// TIA Portal V17 export
// export: Created 2025-03-07T09:17:46.2678876Z, ExportSetting WithDefaults, DisplayName Totally Integrated Automation Portal, DisplayVersion V17 Update 8, DisplayName TIA Portal Openness, DisplayVersion V17 Update 8, DisplayName TIA Portal Version Control Interface, DisplayVersion V17, DisplayName SINAMICS Startdrive Advanced, DisplayVersion V17 SP2, DisplayName SINAMICS Startdrive G110M, G120, G120C, G120D, G120P, G115D, DisplayVersion V17 SP2, DisplayName SINAMICS Startdrive G130, G150, S120, S150, SINAMICS MV, S210, DisplayVersion V17 SP2, DisplayName STEP 7 Professional, DisplayVersion V17 Update 8, DisplayName SINUMERIK ONE STEP 7 Toolbox, DisplayVersion V17 Update 12, DisplayName SINUMERIK 840D sl STEP 7 Toolbox, DisplayVersion V17 Update 12, DisplayName STEP 7 Safety, DisplayVersion V17 Update 6, DisplayName WinCC Advanced, DisplayVersion V17 Update 8
FUNCTION "FC2107_MACHINE_LIGHT" : Void   // FC2107, LAD
{ S7_Optimized_Access := 'FALSE' }
AUTHOR : ETXETAR
VERSION : 1.0
// stored: AutoNumber false, IsIECCheckEnabled false, SetENOAutomatically false, UDAEnableTagReadback false
   VAR_TEMP   // added for the SCL form of the ladder/FBD networks
      _w1 : Bool;
      _w2 : Bool;
      _w3 : Bool;
      _w4 : Bool;
   END_VAR
BEGIN

REGION Network 1: INPUTS
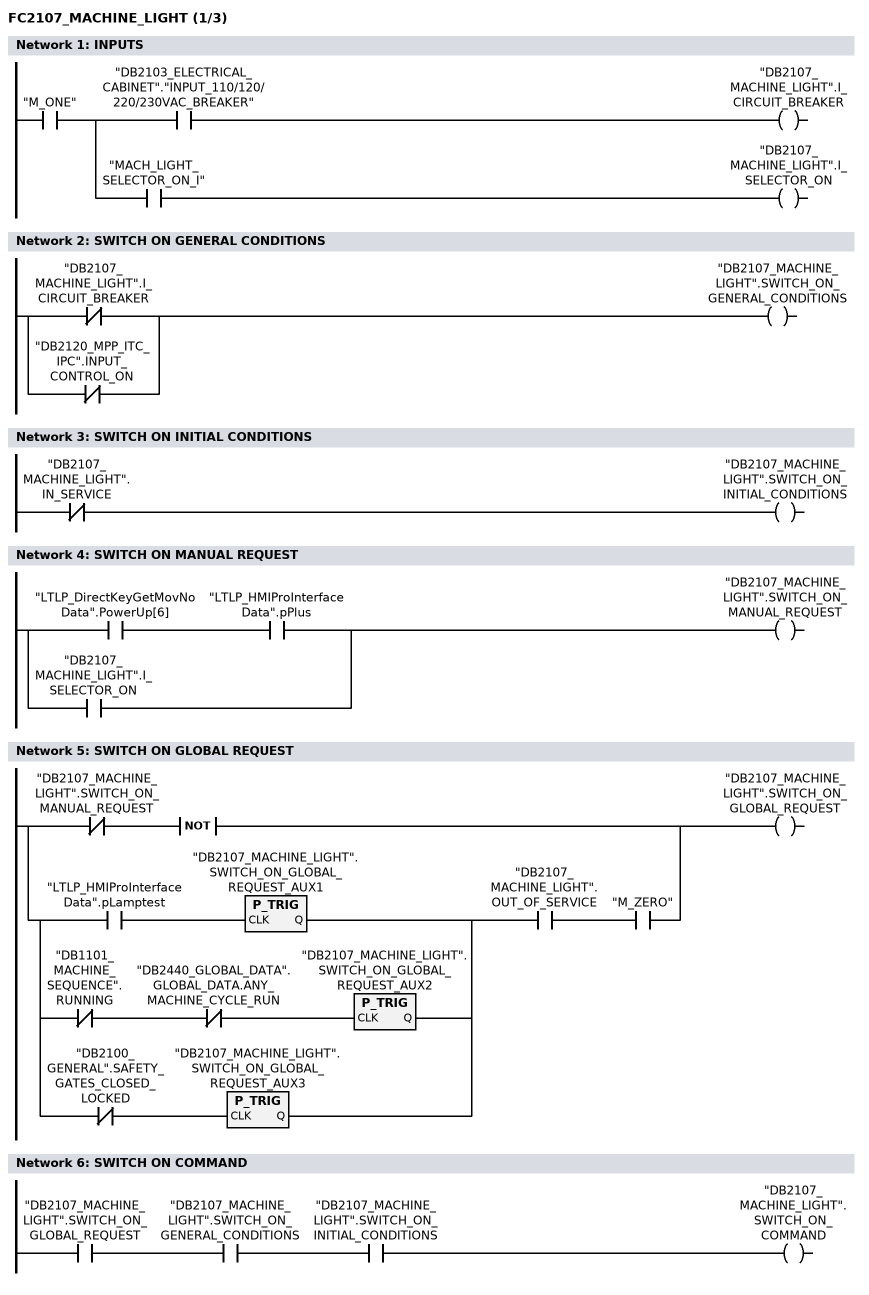
   RUNG wire#powerrail
      Contact( "M_ONE" )
      wire#w1
      Contact( "DB2103_ELECTRICAL_CABINET"."INPUT_110/120/220/230VAC_BREAKER" )
      Coil( "DB2107_MACHINE_LIGHT".I_CIRCUIT_BREAKER )
   END_RUNG
   RUNG wire#w1
      Contact( "MACH_LIGHT_SELECTOR_ON_I" )
      Coil( "DB2107_MACHINE_LIGHT".I_SELECTOR_ON )
   END_RUNG
   // the same network as SCL:
   "DB2107_MACHINE_LIGHT".I_CIRCUIT_BREAKER := "M_ONE" AND "DB2103_ELECTRICAL_CABINET"."INPUT_110/120/220/230VAC_BREAKER";
   "DB2107_MACHINE_LIGHT".I_SELECTOR_ON := "M_ONE" AND "MACH_LIGHT_SELECTOR_ON_I";
END_REGION

REGION Network 2: SWITCH ON GENERAL CONDITIONS
   RUNG wire#powerrail
      I_Contact( "DB2107_MACHINE_LIGHT".I_CIRCUIT_BREAKER )
      wire#w1
      Coil( "DB2107_MACHINE_LIGHT".SWITCH_ON_GENERAL_CONDITIONS )
   END_RUNG
   RUNG wire#powerrail
      I_Contact( "DB2120_MPP_ITC_IPC".INPUT_CONTROL_ON )
   END_RUNG wire#w1
   // the same network as SCL:
   "DB2107_MACHINE_LIGHT".SWITCH_ON_GENERAL_CONDITIONS := NOT "DB2107_MACHINE_LIGHT".I_CIRCUIT_BREAKER OR NOT "DB2120_MPP_ITC_IPC".INPUT_CONTROL_ON;
END_REGION

REGION Network 3: SWITCH ON INITIAL CONDITIONS
   RUNG wire#powerrail
      I_Contact( "DB2107_MACHINE_LIGHT".IN_SERVICE )
      Coil( "DB2107_MACHINE_LIGHT".SWITCH_ON_INITIAL_CONDITIONS )
   END_RUNG
   // the same network as SCL:
   "DB2107_MACHINE_LIGHT".SWITCH_ON_INITIAL_CONDITIONS := NOT "DB2107_MACHINE_LIGHT".IN_SERVICE;
END_REGION

REGION Network 4: SWITCH ON MANUAL REQUEST
   RUNG wire#powerrail
      Contact( "LTLP_DirectKeyGetMovNoData".PowerUp[6] )
      Contact( "LTLP_HMIProInterfaceData".pPlus )
      wire#w1
      Coil( "DB2107_MACHINE_LIGHT".SWITCH_ON_MANUAL_REQUEST )
   END_RUNG
   RUNG wire#powerrail
      Contact( "DB2107_MACHINE_LIGHT".I_SELECTOR_ON )
   END_RUNG wire#w1
   // the same network as SCL:
   "DB2107_MACHINE_LIGHT".SWITCH_ON_MANUAL_REQUEST := ("LTLP_DirectKeyGetMovNoData".PowerUp[6] AND "LTLP_HMIProInterfaceData".pPlus) OR "DB2107_MACHINE_LIGHT".I_SELECTOR_ON;
END_REGION

REGION Network 5: SWITCH ON GLOBAL REQUEST
   RUNG wire#powerrail
      I_Contact( "DB2107_MACHINE_LIGHT".SWITCH_ON_MANUAL_REQUEST )
      Not()
      wire#w1
      Coil( "DB2107_MACHINE_LIGHT".SWITCH_ON_GLOBAL_REQUEST )
   END_RUNG
   RUNG wire#powerrail
      Contact( "LTLP_HMIProInterfaceData".pLamptest )
      P_Trig( "DB2107_MACHINE_LIGHT".SWITCH_ON_GLOBAL_REQUEST_AUX1 )
      wire#w2
      Contact( "DB2107_MACHINE_LIGHT".OUT_OF_SERVICE )
      Contact( "M_ZERO" )
   END_RUNG wire#w1
   RUNG wire#powerrail
      I_Contact( "DB1101_MACHINE_SEQUENCE".RUNNING )
      I_Contact( "DB2440_GLOBAL_DATA".GLOBAL_DATA.ANY_MACHINE_CYCLE_RUN )
      P_Trig( "DB2107_MACHINE_LIGHT".SWITCH_ON_GLOBAL_REQUEST_AUX2 )
   END_RUNG wire#w2
   RUNG wire#powerrail
      I_Contact( "DB2100_GENERAL".SAFETY_GATES_CLOSED_LOCKED )
      P_Trig( "DB2107_MACHINE_LIGHT".SWITCH_ON_GLOBAL_REQUEST_AUX3 )
   END_RUNG wire#w2
   // the same network as SCL:
   #_w1 := "LTLP_HMIProInterfaceData".pLamptest AND NOT "DB2107_MACHINE_LIGHT".SWITCH_ON_GLOBAL_REQUEST_AUX1;   // rising edge
   "DB2107_MACHINE_LIGHT".SWITCH_ON_GLOBAL_REQUEST_AUX1 := "LTLP_HMIProInterfaceData".pLamptest;
   #_w2 := NOT "DB1101_MACHINE_SEQUENCE".RUNNING AND NOT "DB2440_GLOBAL_DATA".GLOBAL_DATA.ANY_MACHINE_CYCLE_RUN;
   #_w3 := #_w2 AND NOT "DB2107_MACHINE_LIGHT".SWITCH_ON_GLOBAL_REQUEST_AUX2;   // rising edge
   "DB2107_MACHINE_LIGHT".SWITCH_ON_GLOBAL_REQUEST_AUX2 := #_w2;
   #_w4 := NOT "DB2100_GENERAL".SAFETY_GATES_CLOSED_LOCKED AND NOT "DB2107_MACHINE_LIGHT".SWITCH_ON_GLOBAL_REQUEST_AUX3;   // rising edge
   "DB2107_MACHINE_LIGHT".SWITCH_ON_GLOBAL_REQUEST_AUX3 := NOT "DB2100_GENERAL".SAFETY_GATES_CLOSED_LOCKED;
   "DB2107_MACHINE_LIGHT".SWITCH_ON_GLOBAL_REQUEST := NOT (NOT "DB2107_MACHINE_LIGHT".SWITCH_ON_MANUAL_REQUEST) OR ((#_w1 OR #_w3 OR #_w4) AND "DB2107_MACHINE_LIGHT".OUT_OF_SERVICE AND "M_ZERO");
END_REGION

REGION Network 6: SWITCH ON COMMAND
   RUNG wire#powerrail
      Contact( "DB2107_MACHINE_LIGHT".SWITCH_ON_GLOBAL_REQUEST )
      Contact( "DB2107_MACHINE_LIGHT".SWITCH_ON_GENERAL_CONDITIONS )
      Contact( "DB2107_MACHINE_LIGHT".SWITCH_ON_INITIAL_CONDITIONS )
      Coil( "DB2107_MACHINE_LIGHT".SWITCH_ON_COMMAND )
   END_RUNG
   // the same network as SCL:
   "DB2107_MACHINE_LIGHT".SWITCH_ON_COMMAND := "DB2107_MACHINE_LIGHT".SWITCH_ON_GLOBAL_REQUEST AND "DB2107_MACHINE_LIGHT".SWITCH_ON_GENERAL_CONDITIONS AND "DB2107_MACHINE_LIGHT".SWITCH_ON_INITIAL_CONDITIONS;
END_REGION

REGION Network 7: SWITCH ON
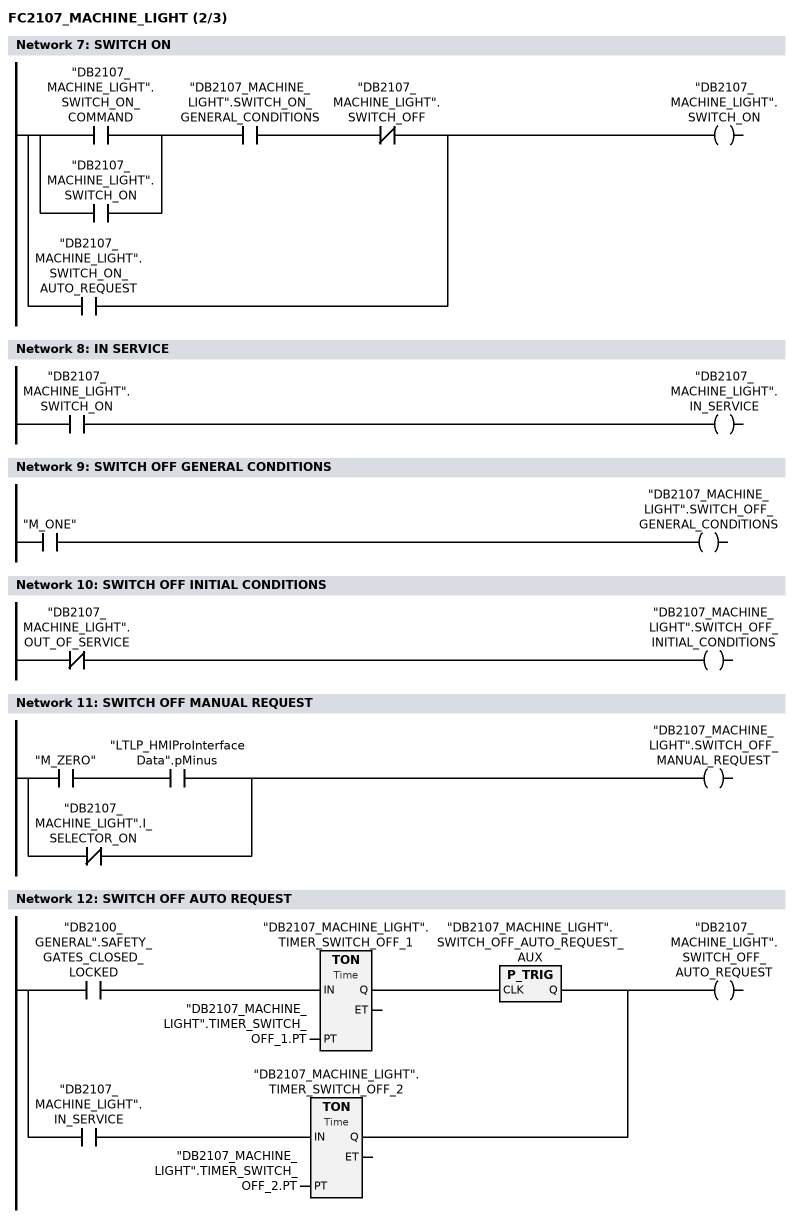
   RUNG wire#powerrail
      Contact( "DB2107_MACHINE_LIGHT".SWITCH_ON_COMMAND )
      wire#w1
      Contact( "DB2107_MACHINE_LIGHT".SWITCH_ON_GENERAL_CONDITIONS )
      I_Contact( "DB2107_MACHINE_LIGHT".SWITCH_OFF )
      wire#w2
      Coil( "DB2107_MACHINE_LIGHT".SWITCH_ON )
   END_RUNG
   RUNG wire#powerrail
      Contact( "DB2107_MACHINE_LIGHT".SWITCH_ON )
   END_RUNG wire#w1
   RUNG wire#powerrail
      Contact( "DB2107_MACHINE_LIGHT".SWITCH_ON_AUTO_REQUEST )
   END_RUNG wire#w2
   // the same network as SCL:
   "DB2107_MACHINE_LIGHT".SWITCH_ON := (("DB2107_MACHINE_LIGHT".SWITCH_ON_COMMAND OR "DB2107_MACHINE_LIGHT".SWITCH_ON) AND "DB2107_MACHINE_LIGHT".SWITCH_ON_GENERAL_CONDITIONS AND NOT "DB2107_MACHINE_LIGHT".SWITCH_OFF) OR "DB2107_MACHINE_LIGHT".SWITCH_ON_AUTO_REQUEST;
END_REGION

REGION Network 8: IN SERVICE
   RUNG wire#powerrail
      Contact( "DB2107_MACHINE_LIGHT".SWITCH_ON )
      Coil( "DB2107_MACHINE_LIGHT".IN_SERVICE )
   END_RUNG
   // the same network as SCL:
   "DB2107_MACHINE_LIGHT".IN_SERVICE := "DB2107_MACHINE_LIGHT".SWITCH_ON;
END_REGION

REGION Network 9: SWITCH OFF GENERAL CONDITIONS
   RUNG wire#powerrail
      Contact( "M_ONE" )
      Coil( "DB2107_MACHINE_LIGHT".SWITCH_OFF_GENERAL_CONDITIONS )
   END_RUNG
   // the same network as SCL:
   "DB2107_MACHINE_LIGHT".SWITCH_OFF_GENERAL_CONDITIONS := "M_ONE";
END_REGION

REGION Network 10: SWITCH OFF INITIAL CONDITIONS
   RUNG wire#powerrail
      I_Contact( "DB2107_MACHINE_LIGHT".OUT_OF_SERVICE )
      Coil( "DB2107_MACHINE_LIGHT".SWITCH_OFF_INITIAL_CONDITIONS )
   END_RUNG
   // the same network as SCL:
   "DB2107_MACHINE_LIGHT".SWITCH_OFF_INITIAL_CONDITIONS := NOT "DB2107_MACHINE_LIGHT".OUT_OF_SERVICE;
END_REGION

REGION Network 11: SWITCH OFF MANUAL REQUEST
   RUNG wire#powerrail
      Contact( "M_ZERO" )
      Contact( "LTLP_HMIProInterfaceData".pMinus )
      wire#w1
      Coil( "DB2107_MACHINE_LIGHT".SWITCH_OFF_MANUAL_REQUEST )
   END_RUNG
   RUNG wire#powerrail
      I_Contact( "DB2107_MACHINE_LIGHT".I_SELECTOR_ON )
   END_RUNG wire#w1
   // the same network as SCL:
   "DB2107_MACHINE_LIGHT".SWITCH_OFF_MANUAL_REQUEST := ("M_ZERO" AND "LTLP_HMIProInterfaceData".pMinus) OR NOT "DB2107_MACHINE_LIGHT".I_SELECTOR_ON;
END_REGION

REGION Network 12: SWITCH OFF AUTO REQUEST
   RUNG wire#powerrail
      Contact( "DB2100_GENERAL".SAFETY_GATES_CLOSED_LOCKED )
      { S7_Templates := "time_type := Time" } "DB2107_MACHINE_LIGHT".TIMER_SWITCH_OFF_1.TON(pt := "DB2107_MACHINE_LIGHT".TIMER_SWITCH_OFF_1.PT, et =>)
      P_Trig( "DB2107_MACHINE_LIGHT".SWITCH_OFF_AUTO_REQUEST_AUX )
      wire#w1
      Coil( "DB2107_MACHINE_LIGHT".SWITCH_OFF_AUTO_REQUEST )
   END_RUNG
   RUNG wire#powerrail
      Contact( "DB2107_MACHINE_LIGHT".IN_SERVICE )
      { S7_Templates := "time_type := Time" } "DB2107_MACHINE_LIGHT".TIMER_SWITCH_OFF_2.TON(pt := "DB2107_MACHINE_LIGHT".TIMER_SWITCH_OFF_2.PT, et =>)
   END_RUNG wire#w1
   // the same network as SCL:
   "DB2107_MACHINE_LIGHT".TIMER_SWITCH_OFF_1.TON(IN := "DB2100_GENERAL".SAFETY_GATES_CLOSED_LOCKED,
                           PT := "DB2107_MACHINE_LIGHT".TIMER_SWITCH_OFF_1.PT);
   #_w1 := "DB2107_MACHINE_LIGHT".TIMER_SWITCH_OFF_1.Q AND NOT "DB2107_MACHINE_LIGHT".SWITCH_OFF_AUTO_REQUEST_AUX;   // rising edge
   "DB2107_MACHINE_LIGHT".SWITCH_OFF_AUTO_REQUEST_AUX := "DB2107_MACHINE_LIGHT".TIMER_SWITCH_OFF_1.Q;
   "DB2107_MACHINE_LIGHT".TIMER_SWITCH_OFF_2.TON(IN := "DB2107_MACHINE_LIGHT".IN_SERVICE,
                           PT := "DB2107_MACHINE_LIGHT".TIMER_SWITCH_OFF_2.PT);
   "DB2107_MACHINE_LIGHT".SWITCH_OFF_AUTO_REQUEST := #_w1 OR "DB2107_MACHINE_LIGHT".TIMER_SWITCH_OFF_2.Q;
END_REGION

REGION Network 13: SWITCH OFF GLOBAL REQUEST
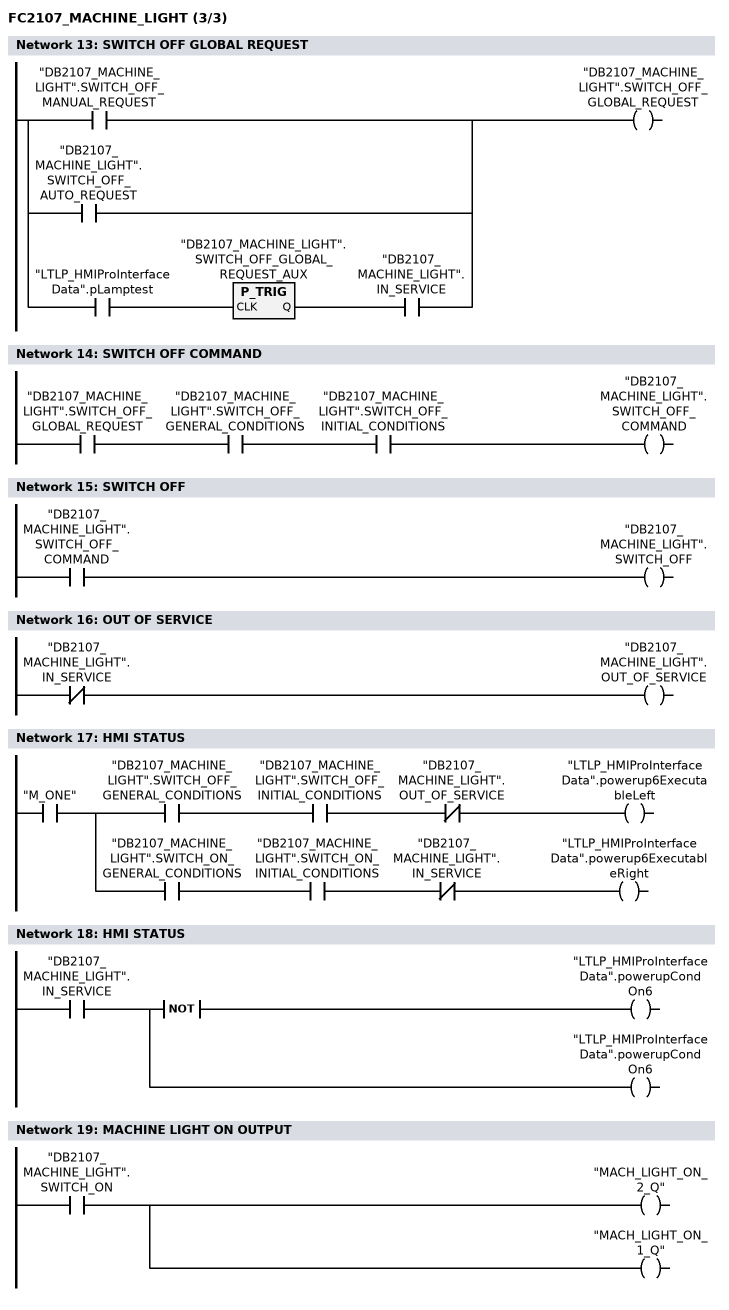
   RUNG wire#powerrail
      Contact( "DB2107_MACHINE_LIGHT".SWITCH_OFF_MANUAL_REQUEST )
      wire#w1
      Coil( "DB2107_MACHINE_LIGHT".SWITCH_OFF_GLOBAL_REQUEST )
   END_RUNG
   RUNG wire#powerrail
      Contact( "DB2107_MACHINE_LIGHT".SWITCH_OFF_AUTO_REQUEST )
   END_RUNG wire#w1
   RUNG wire#powerrail
      Contact( "LTLP_HMIProInterfaceData".pLamptest )
      P_Trig( "DB2107_MACHINE_LIGHT".SWITCH_OFF_GLOBAL_REQUEST_AUX )
      Contact( "DB2107_MACHINE_LIGHT".IN_SERVICE )
   END_RUNG wire#w1
   // the same network as SCL:
   #_w1 := "LTLP_HMIProInterfaceData".pLamptest AND NOT "DB2107_MACHINE_LIGHT".SWITCH_OFF_GLOBAL_REQUEST_AUX;   // rising edge
   "DB2107_MACHINE_LIGHT".SWITCH_OFF_GLOBAL_REQUEST_AUX := "LTLP_HMIProInterfaceData".pLamptest;
   "DB2107_MACHINE_LIGHT".SWITCH_OFF_GLOBAL_REQUEST := "DB2107_MACHINE_LIGHT".SWITCH_OFF_MANUAL_REQUEST OR "DB2107_MACHINE_LIGHT".SWITCH_OFF_AUTO_REQUEST OR (#_w1 AND "DB2107_MACHINE_LIGHT".IN_SERVICE);
END_REGION

REGION Network 14: SWITCH OFF COMMAND
   RUNG wire#powerrail
      Contact( "DB2107_MACHINE_LIGHT".SWITCH_OFF_GLOBAL_REQUEST )
      Contact( "DB2107_MACHINE_LIGHT".SWITCH_OFF_GENERAL_CONDITIONS )
      Contact( "DB2107_MACHINE_LIGHT".SWITCH_OFF_INITIAL_CONDITIONS )
      Coil( "DB2107_MACHINE_LIGHT".SWITCH_OFF_COMMAND )
   END_RUNG
   // the same network as SCL:
   "DB2107_MACHINE_LIGHT".SWITCH_OFF_COMMAND := "DB2107_MACHINE_LIGHT".SWITCH_OFF_GLOBAL_REQUEST AND "DB2107_MACHINE_LIGHT".SWITCH_OFF_GENERAL_CONDITIONS AND "DB2107_MACHINE_LIGHT".SWITCH_OFF_INITIAL_CONDITIONS;
END_REGION

REGION Network 15: SWITCH OFF
   RUNG wire#powerrail
      Contact( "DB2107_MACHINE_LIGHT".SWITCH_OFF_COMMAND )
      Coil( "DB2107_MACHINE_LIGHT".SWITCH_OFF )
   END_RUNG
   // the same network as SCL:
   "DB2107_MACHINE_LIGHT".SWITCH_OFF := "DB2107_MACHINE_LIGHT".SWITCH_OFF_COMMAND;
END_REGION

REGION Network 16: OUT OF SERVICE
   RUNG wire#powerrail
      I_Contact( "DB2107_MACHINE_LIGHT".IN_SERVICE )
      Coil( "DB2107_MACHINE_LIGHT".OUT_OF_SERVICE )
   END_RUNG
   // the same network as SCL:
   "DB2107_MACHINE_LIGHT".OUT_OF_SERVICE := NOT "DB2107_MACHINE_LIGHT".IN_SERVICE;
END_REGION

REGION Network 17: HMI STATUS
   RUNG wire#powerrail
      Contact( "M_ONE" )
      wire#w1
      Contact( "DB2107_MACHINE_LIGHT".SWITCH_OFF_GENERAL_CONDITIONS )
      Contact( "DB2107_MACHINE_LIGHT".SWITCH_OFF_INITIAL_CONDITIONS )
      I_Contact( "DB2107_MACHINE_LIGHT".OUT_OF_SERVICE )
      Coil( "LTLP_HMIProInterfaceData".powerup6ExecutableLeft )
   END_RUNG
   RUNG wire#w1
      Contact( "DB2107_MACHINE_LIGHT".SWITCH_ON_GENERAL_CONDITIONS )
      Contact( "DB2107_MACHINE_LIGHT".SWITCH_ON_INITIAL_CONDITIONS )
      I_Contact( "DB2107_MACHINE_LIGHT".IN_SERVICE )
      Coil( "LTLP_HMIProInterfaceData".powerup6ExecutableRight )
   END_RUNG
   // the same network as SCL:
   "LTLP_HMIProInterfaceData".powerup6ExecutableLeft := "M_ONE" AND "DB2107_MACHINE_LIGHT".SWITCH_OFF_GENERAL_CONDITIONS AND "DB2107_MACHINE_LIGHT".SWITCH_OFF_INITIAL_CONDITIONS AND NOT "DB2107_MACHINE_LIGHT".OUT_OF_SERVICE;
   "LTLP_HMIProInterfaceData".powerup6ExecutableRight := "M_ONE" AND "DB2107_MACHINE_LIGHT".SWITCH_ON_GENERAL_CONDITIONS AND "DB2107_MACHINE_LIGHT".SWITCH_ON_INITIAL_CONDITIONS AND NOT "DB2107_MACHINE_LIGHT".IN_SERVICE;
END_REGION

REGION Network 18: HMI STATUS
   RUNG wire#powerrail
      Contact( "DB2107_MACHINE_LIGHT".IN_SERVICE )
      wire#w1
      Not()
      Coil( "LTLP_HMIProInterfaceData".powerupCondOn6 )
   END_RUNG
   RUNG wire#w1
      Coil( "LTLP_HMIProInterfaceData".powerupCondOn6 )
   END_RUNG
   // the same network as SCL:
   "LTLP_HMIProInterfaceData".powerupCondOn6 := NOT "DB2107_MACHINE_LIGHT".IN_SERVICE;
   "LTLP_HMIProInterfaceData".powerupCondOn6 := "DB2107_MACHINE_LIGHT".IN_SERVICE;
END_REGION

REGION Network 19: MACHINE LIGHT ON OUTPUT
   RUNG wire#powerrail
      Contact( "DB2107_MACHINE_LIGHT".SWITCH_ON )
      wire#w1
      Coil( "MACH_LIGHT_ON_2_Q" )
   END_RUNG
   RUNG wire#w1
      Coil( "MACH_LIGHT_ON_1_Q" )
   END_RUNG
   // the same network as SCL:
   "MACH_LIGHT_ON_2_Q" := "DB2107_MACHINE_LIGHT".SWITCH_ON;
   "MACH_LIGHT_ON_1_Q" := "DB2107_MACHINE_LIGHT".SWITCH_ON;
END_REGION
END_FUNCTION
